{attribute 'qualified_only'}
{attribute 'strict'}
TYPE E_CalibStep :
(
	IDLE 				:= 0, 	// Idle State
    DELAY 				:= 5, 	// Delay state depending on delay time to start calibration on HMI
	CHECKING_WEIGH 		:= 10,	// Checking if the calibration box is on the correct weight
	POSITION_MOTORS 	:= 20,	// Position the motors M2 and M3 to calibration position
	POSITION_VALVES 	:= 30,	// Position Valves into calibration position
	FILLJAR_FORWARD 	:= 40,	// Fill the jars first with the volume in the HMI plus tubing dead volume
	WEIGH_BEFORE 		:= 50,	// Request calibration box weight [Tare weight]
	WITHDRAW_BACKWARDS 	:= 60,	// Pump back to calibration box the amount of liquid into the HMI
	WEIGH_AFTER 		:= 70,	// Request the calibration box weight after pumping [Gross Weight]  
	RETURN_FORWARD 		:= 80,	// Return to the jar the same amount of liquid that was dosed by the pump
	PUMPFACTOR_ADJUST	:= 85,	// Adjust the pump factor if the net volume is less than 10% off the target 
	PUMPFACTOR_FAILED	:= 86,	// If pump factor number of adjustments is greater than allowable failures
	FEED_HMI_RESULTS	:= 90,  // Feed HMI controls with pump results 
	EMPTYJAR_BACKWARDS 	:= 95,	// Empty the Jar with 60% more revs to make sure everything was cleaned
	NEXT_PUMP 			:= 100,	// Going to next pump calibration
	HOMING_MOTORS 		:= 110,	// Moving the motors M2 and M3 back to home position
	REPORT_INFO_UPDATE	:= 120, // Step where all the reports info are updated
	AIR_DRY_TIME		:= 130, // Air Dry Time when calibration is finished
	CALBOX_ATTENTION	:= 170, // Step where the FB waits for someone fill up the calibration box
	SCALE_ATTENTION		:= 180, // Step where the FB waits for human interaction in the scale
	COMPLETE 			:= 200,	// Complete state
	ERROR 				:= 300	// Error state
);
END_TYPE

(* stored: Version 1.1.0.1, ProductVersion 3.1.4024.15
   DUT E_CalibStep: Id {5a17fee5-548f-4ae8-9c80-2b454d06d508} *)
